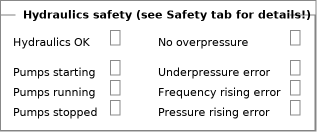
VISUALIZATION VISU_HydraulicsSafety  // 317x132
VAR_IN_OUT
	ref : Hydraulics;
    widget : HydraulicsWidget;
    ref_safety : SafetyHydraulics;
END_VAR
    Polyline (15,15) (0,15) (0,130) (315,130) (315,15) (290,15)
    Label (20,5 270x20), "Hydraulics safety (see Safety tab for details!)"
    Label (10,30 95x25), "Hydraulics OK"
    Frame (110,30 10x15)
        shows VISU_State_red_green(state := ref_safety.allOK)
    Label (10,60 95x25), "Pumps starting"
    Frame (110,60 10x15)
        shows VISU_State_gray_green(state := ref_safety.pumpsStartingUp)
    Label (10,80 95x25), "Pumps running"
    Frame (110,80 10x15)
        shows VISU_State_gray_green(state := ref_safety.pumpsRunning)
    Label (10,100 95x25), "Pumps stopped"
    Frame (110,100 10x15)
        shows VISU_State_gray_green(state := ref_safety.pumpsStopped)
    Label (155,30 120x25), "No overpressure"
    Frame (290,30 10x15)
        shows VISU_State_gray_green(state := ref_safety.noOverpressure)
    Label (155,60 120x25), "Underpressure error"
    Frame (290,60 10x15)
        shows VISU_State_gray_red(state := ref_safety.underpressureError)
    Label (155,80 130x25), "Frequency rising error"
    Frame (290,80 10x15)
        shows VISU_State_gray_red(state := ref_safety.pumpsFrequencyNotRising)
    Label (155,100 130x25), "Pressure rising error"
    Frame (290,100 10x15)
        shows VISU_State_gray_red(state := ref_safety.pressureNotRising)
END_VISUALIZATION

(* stored: Version 1.1.0.1, ProductVersion 3.1.4019.2
   Visu VISU_HydraulicsSafety: Id {09c56ffc-1738-46be-aea6-d4a7e5a957df} *)
